// TIA Portal V18 export
DATA_BLOCK "Call_KeyenceCheckerIV_DB"   // DB2100
// stored: AutoNumber false, InstanceOfName Call_KeyenceCheckerIV, InstanceOfType FB
"Call_KeyenceCheckerIV"
   // VAR
   //    InsKeyenceCheckerIV3810A1 : "FB_KeyenceCheckerIV3";
   //    InsKeyenceCheckerIV3811A1 : "FB_KeyenceCheckerIV3";
   //    nIndex { S7_SetPoint := 'True'} : Int;
   // END_VAR
BEGIN
END_DATA_BLOCK
